PROGRAM MAIN
VAR
	stEventsMain : ST_Events;
	xFlag :   BOOL := FALSE;
END_VAR

IF NOT xFlag THEN
		F_UpdateTimestamp (stEventsMain);
		xFlag := TRUE;
END_IF

END_PROGRAM

(* stored: Version 1.1.0.1, ProductVersion 3.1.4024.11
   POU MAIN: Id {13015835-c886-43a5-a180-937f16083639}, SpecialFunc None *)
